(* CoDeSys 2.3.9.31 project: convertedProject.pr6 *)
(* Libraries: Standard.lib 5.6.98 11:03:02 *)

(* Task configuration *)
TASK MainTask (PRIORITY := 1, INTERVAL := T#200ms);
	MAIN();
END_TASK

(* Global variable list: Global_Variables *)
VAR_GLOBAL
	(* Контроль 0 *)
	G_IN_CTL_BTN_1: BOOL; (* Кнопка ALL *)
	G_IN_CTL_BTN_2: BOOL; (* Кнопка RESET *)
	G_OUT_CTL_ALARM_LAMP: BOOL; (* Лампа-сигнализатор *)
	G_OUT_CTL_ALARM_SOUND: BOOL; (* Динамик в ПЛК *)
	G_OUT_CTL_SOCKET_1: BOOL; (* Питание для МВВ *)

	(* Дверь *)
	G_IN_DOOR_DTR_1: BOOL; (* Сенсор открытия двери *)
	G_IN_DOOR_BTN_BELL: BOOL; (* Кнопка звонка *)
	G_OUT_DOOR_BELL: BOOL; (* Звонок *)

	(* Кухня 1 *)
	G_IN_KTN_BTN_1: BOOL; (* Выключатель основной *)
	G_IN_KTN_BTN_2: BOOL; (* Выключатель для вытяжки *)
	G_IN_KTN_DTR_1: BOOL; (* Датчик протечек *)
	G_OUT_KTN_LIGHT_1: BOOL; (* Свет основной *)
	G_OUT_KTN_LIGHT_2: BOOL; (* Свет второстепенный (подсветка) *)
	G_OUT_KTN_FAN_1: BOOL; (* Вытяжка *)

	(* Балкон *)
	G_IN_BLKN_BTN_1: BOOL; (* Выключатель *)
	G_OUT_BLKN_LIGHT_1: BOOL; (* Свет *)

	(* Гостиная *)
	G_IN_LVG_BTN_1: BOOL; (* Выключатель *)
	G_IN_LVG_BTN_2: BOOL; (* Выключатель на рабочем месте *)
	G_OUT_LVG_LIGHT_1: BOOL; (* Свет основной *)
	G_OUT_LVG_LIGHT_2: BOOL; (* Свет второстепенный *)

	(* Спальная *)
	G_IN_BDR_BTN_1: BOOL; (* Выключатель *)
	G_IN_BDR_BTN_2: BOOL; (* Выключатель над кроватью *)
	G_IN_BDR_BTN_3: BOOL; (* Выключатель над кроватью *)
	G_OUT_BDR_LIGHT_1: BOOL; (* Свет *)
	G_OUT_BDR_LIGHT_2: BOOL; (* Свет второстепенный *)
	G_OUT_BDR_LIGHT_3: BOOL; (* Свет над кроватью (торшер) *)
	G_OUT_BDR_LIGHT_4: BOOL; (* Свет над кроватью (торшер) *)

	(* Ванная большая *)
	G_IN_BMB_BTN_1: BOOL; (* Выключатель основной *)
	G_IN_BMB_BTN_2: BOOL; (* Выключатель около зеркала *)
	G_IN_BMB_DTR_1: BOOL; (* Датчик протечек *)
	G_OUT_BMB_LIGHT_1: BOOL; (* Свет основной *)
	G_OUT_BMB_LIGHT_2: BOOL; (* Свет около зеркала *)
	G_OUT_BMB_FAN_1: BOOL; (* Вытяжка *)
	G_OUT_BMB_VLV_1: BOOL; (* Вентиль *)
	G_OUT_BMB_VLV_2: BOOL; (* Вентиль *)

	(* Детская *)
	G_IN_CHLD_BTN_1: BOOL; (* Выключатель *)
	G_OUT_CHLD_LIGHT_1: BOOL; (* Свет основной *)
	G_OUT_CHLD_LIGHT_2: BOOL; (* Свет второстепенный *)

	(* Коридор *)
	G_IN_HLL_BTN_1: BOOL; (* Проходной выключатель *)
	G_IN_HLL_BTN_2: BOOL; (* Проходной выключатель *)
	G_IN_HLL_BTN_3: BOOL; (* Выключатель на зеркало *)
	G_IN_HLL_BTN_4: BOOL; (* Выключатель в шкафу *)
	G_IN_HLL_BTN_5: BOOL; (* Выключатель в шкафу *)

	G_OUT_HLL_LIGHT_1: BOOL; (* Свет основной *)
	G_OUT_HLL_LIGHT_2: BOOL; (* Свет второстепенный *)
	G_OUT_HLL_LIGHT_3: BOOL; (* Свет зеркало *)
	G_OUT_HLL_LIGHT_4: BOOL; (* Свет в шкафу *)
	G_OUT_HLL_LIGHT_5: BOOL; (* Свет в шкафу *)

	(* Ванная малая *)
	G_IN_BMS_BTN_1: BOOL; (* Выключатель *)
	G_IN_BMS_DTR_1: BOOL; (* Датчик протечек *)
	G_OUT_BMS_LIGHT_1: BOOL; (* Вытяжка *)
	G_OUT_BMS_FAN_1: BOOL; (* Вытяжка *)
	G_OUT_BMS_VLV_1: BOOL; (* Вентиль *)
	G_OUT_BMS_VLV_2: BOOL; (* Вентиль *)

	(* Розетки *)
	(* Кухня и балкон *)
	G_OUT_1_2_SOCKET_G1: BOOL; (* Общие *)
	G_OUT_1_2_SOCKET_G2: BOOL; (* Неотключаемые (холодильник)*)
	G_OUT_1_2_SOCKET_G3: BOOL; (* Посудомойка *)
	G_OUT_1_2_SOCKET_G4: BOOL; (* Плита, 380В *)
	(* Гостиная и спальня *)
	G_OUT_3_4_SOCKET_G1: BOOL; (* Общие *)
	G_OUT_3_4_SOCKET_G2: BOOL; (* Неотключаемые (компьютер) *)
	(* Ванная большая *)
	G_OUT_5_SOCKET_G1: BOOL; (* Общие *)
	G_OUT_5_SOCKET_G2: BOOL; (* Стиральная машина *)
	G_OUT_5_SOCKET_G3: BOOL; (* Резерв на бойлер и (или) баню *)
	(* Коридор и детская *)
	G_OUT_6_7_SOCKET_G1: BOOL; (* Общие *)
	G_OUT_6_7_SOCKET_G2: BOOL; (* Неотключаемые (рядом со щитком, роутер, сервер и т.п.) *)

END_VAR

(* Global variable list: TwinCAT_Import *)
VAR_GLOBAL (* DO NOT CHANGE THIS SHEET MANUALLY! *)
	PlcInVar_0	AT %QB128:	USINT;
	PlcInVar_1	AT %QB129:	USINT;
	PlcInVar_2	AT %QB130:	USINT;
	PlcInVar_3	AT %QB131:	USINT;
	PlcInVar_4	AT %QB132:	USINT;
	PlcInVar_5	AT %QB133:	USINT;
	PlcInVar_6	AT %QB134:	USINT;
	PlcInVar_7	AT %QB135:	USINT;
	PlcInVar_8	AT %QB136:	USINT;
	PlcInVar_9	AT %QB137:	USINT;
	PlcInVar_10	AT %QB138:	USINT;
	PlcInVar_11	AT %QB139:	USINT;
	PlcInVar_12	AT %QB140:	USINT;
	PlcInVar_13	AT %QB141:	USINT;
	PlcInVar_14	AT %QB142:	USINT;
	PlcInVar_15	AT %QB143:	USINT;
	PlcOutVar_0	AT %IB128:	USINT;
	PlcOutVar_1	AT %IB129:	USINT;
	PlcOutVar_2	AT %IB130:	USINT;
	PlcOutVar_3	AT %IB131:	USINT;
	PlcOutVar_4	AT %IB132:	USINT;
	PlcOutVar_5	AT %IB133:	USINT;
	PlcOutVar_6	AT %IB134:	USINT;
	PlcOutVar_7	AT %IB135:	USINT;
	PlcOutVar_8	AT %IB136:	USINT;
	PlcOutVar_9	AT %IB137:	USINT;
	PlcOutVar_10	AT %IB138:	USINT;
	PlcOutVar_11	AT %IB139:	USINT;
	PlcOutVar_12	AT %IB140:	USINT;
	PlcOutVar_13	AT %IB141:	USINT;
	PlcOutVar_14	AT %IB142:	USINT;
	PlcOutVar_15	AT %IB143:	USINT;
	Term_2_KL2408_1_Output	AT %QX0.0:	BOOL;
	Term_2_KL2408_2_Output	AT %QX0.1:	BOOL;
	Term_2_KL2408_3_Output	AT %QX0.2:	BOOL;
	Term_2_KL2408_4_Output	AT %QX0.3:	BOOL;
	Term_2_KL2408_5_Output	AT %QX0.4:	BOOL;
	Term_2_KL2408_6_Output	AT %QX0.5:	BOOL;
	Term_2_KL2408_7_Output	AT %QX0.6:	BOOL;
	Term_2_KL2408_8_Output	AT %QX0.7:	BOOL;
	Term_3_KL2408_1_Output	AT %QX1.0:	BOOL;
	Term_3_KL2408_2_Output	AT %QX1.1:	BOOL;
	Term_3_KL2408_3_Output	AT %QX1.2:	BOOL;
	Term_3_KL2408_4_Output	AT %QX1.3:	BOOL;
	Term_3_KL2408_5_Output	AT %QX1.4:	BOOL;
	Term_3_KL2408_6_Output	AT %QX1.5:	BOOL;
	Term_3_KL2408_7_Output	AT %QX1.6:	BOOL;
	Term_3_KL2408_8_Output	AT %QX1.7:	BOOL;
	Term_4_KL2408_1_Output	AT %QX2.0:	BOOL;
	Term_4_KL2408_2_Output	AT %QX2.1:	BOOL;
	Term_4_KL2408_3_Output	AT %QX2.2:	BOOL;
	Term_4_KL2408_4_Output	AT %QX2.3:	BOOL;
	Term_4_KL2408_5_Output	AT %QX2.4:	BOOL;
	Term_4_KL2408_6_Output	AT %QX2.5:	BOOL;
	Term_4_KL2408_7_Output	AT %QX2.6:	BOOL;
	Term_4_KL2408_8_Output	AT %QX2.7:	BOOL;
	Term_5_KL2408_1_Output	AT %QX3.0:	BOOL;
	Term_5_KL2408_2_Output	AT %QX3.1:	BOOL;
	Term_5_KL2408_3_Output	AT %QX3.2:	BOOL;
	Term_5_KL2408_4_Output	AT %QX3.3:	BOOL;
	Term_5_KL2408_5_Output	AT %QX3.4:	BOOL;
	Term_5_KL2408_6_Output	AT %QX3.5:	BOOL;
	Term_5_KL2408_7_Output	AT %QX3.6:	BOOL;
	Term_5_KL2408_8_Output	AT %QX3.7:	BOOL;
	Term_6_KL2408_1_Output	AT %QX4.0:	BOOL;
	Term_6_KL2408_2_Output	AT %QX4.1:	BOOL;
	Term_6_KL2408_3_Output	AT %QX4.2:	BOOL;
	Term_6_KL2408_4_Output	AT %QX4.3:	BOOL;
	Term_6_KL2408_5_Output	AT %QX4.4:	BOOL;
	Term_6_KL2408_6_Output	AT %QX4.5:	BOOL;
	Term_6_KL2408_7_Output	AT %QX4.6:	BOOL;
	Term_6_KL2408_8_Output	AT %QX4.7:	BOOL;
	Term_7_KL1408_1_Input	AT %IX0.0:	BOOL;
	Term_7_KL1408_2_Input	AT %IX0.1:	BOOL;
	Term_7_KL1408_3_Input	AT %IX0.2:	BOOL;
	Term_7_KL1408_4_Input	AT %IX0.3:	BOOL;
	Term_7_KL1408_5_Input	AT %IX0.4:	BOOL;
	Term_7_KL1408_6_Input	AT %IX0.5:	BOOL;
	Term_7_KL1408_7_Input	AT %IX0.6:	BOOL;
	Term_7_KL1408_8_Input	AT %IX0.7:	BOOL;
	Term_8_KL1408_1_Input	AT %IX1.0:	BOOL;
	Term_8_KL1408_2_Input	AT %IX1.1:	BOOL;
	Term_8_KL1408_3_Input	AT %IX1.2:	BOOL;
	Term_8_KL1408_4_Input	AT %IX1.3:	BOOL;
	Term_8_KL1408_5_Input	AT %IX1.4:	BOOL;
	Term_8_KL1408_6_Input	AT %IX1.5:	BOOL;
	Term_8_KL1408_7_Input	AT %IX1.6:	BOOL;
	Term_8_KL1408_8_Input	AT %IX1.7:	BOOL;
	Term_9_KL1408_1_Input	AT %IX2.0:	BOOL;
	Term_9_KL1408_2_Input	AT %IX2.1:	BOOL;
	Term_9_KL1408_3_Input	AT %IX2.2:	BOOL;
	Term_9_KL1408_4_Input	AT %IX2.3:	BOOL;
	Term_9_KL1408_5_Input	AT %IX2.4:	BOOL;
	Term_9_KL1408_6_Input	AT %IX2.5:	BOOL;
	Term_9_KL1408_7_Input	AT %IX2.6:	BOOL;
	Term_9_KL1408_8_Input	AT %IX2.7:	BOOL;
	Term_10_KL1408_1_Input	AT %IX3.0:	BOOL;
	Term_10_KL1408_2_Input	AT %IX3.1:	BOOL;
	Term_10_KL1408_3_Input	AT %IX3.2:	BOOL;
	Term_10_KL1408_4_Input	AT %IX3.3:	BOOL;
	Term_10_KL1408_5_Input	AT %IX3.4:	BOOL;
	Term_10_KL1408_6_Input	AT %IX3.5:	BOOL;
	Term_10_KL1408_7_Input	AT %IX3.6:	BOOL;
	Term_10_KL1408_8_Input	AT %IX3.7:	BOOL;
END_VAR

(* POU MAIN, ST *)
PROGRAM MAIN
VAR
	KTN_BTN_1 : Z_FB_DIFF_OUT_ON_LONG_AND_SHORT;
	KTN_BTN_2 : Z_FB_SINGLE_SW;

	BLKN_BTN : Z_FB_SINGLE_SW;

	LVG_BTN : Z_FB_SHORT_P_OUT1_LONG_P_OUT1_AND_OUT2;

	BDR_BTN_1 : Z_FB_SHORT_P_OUT1_LONG_P_OUT1_AND_OUT2;
	BDR_BTN_2 : Z_FB_SINGLE_SW;
	BDR_BTN_3 : Z_FB_SINGLE_SW;

	BMB_BTN_1 : Z_FB_SHRT_P_OUT1_LNG_P_OUT1_OUT2_TIMER;
	BMB_BTN_2 : Z_FB_SINGLE_SW;

	CHLD_BTN : Z_FB_SHORT_P_OUT1_LONG_P_OUT1_AND_OUT2;

	HLL_BTN_1_2 : FB_HLL;
	HLL_BTN_3 : Z_FB_SINGLE_SW_WITH_TIMER;
	HLL_BTN_4 : Z_FB_SINGLE_SW_WITH_TIMER;
	HLL_BTN_5 : Z_FB_SINGLE_SW_WITH_TIMER;

	BMS_BTN : Z_FB_SHRT_P_OUT1_LNG_P_OUT1_OUT2_TIMER;

	CTL_BTN_ALL : FB_ALL;

	IN_WS_LEFT : Z_FB_WS;
	IN_WS_RIGHT : Z_FB_WS;

	T_LONG_PRESS : TIME := t#1000ms;
	T_LIGHT_OFF : TIME := t#5000ms;
	T_FAN_OFF : TIME := t#5000ms;

	ALARM : FB_ALARM;

	ERROR : BOOL;

END_VAR
(* Основной выключатель на кухне *)
KTN_BTN_1 (IN := G_IN_KTN_BTN_1, Q1 := G_OUT_KTN_LIGHT_1, Q2 := G_OUT_KTN_LIGHT_2, TC := T_LONG_PRESS);

(* Второстепенный выключатель на кухне *)
KTN_BTN_2 (IN := G_IN_KTN_BTN_2, Q :=  G_OUT_KTN_FAN_1);

(* Выключатель на балконе *)
BLKN_BTN (IN := G_IN_BLKN_BTN_1, Q := G_OUT_BLKN_LIGHT_1);

(* Выключатели в гостиной *)
LVG_BTN (IN := G_IN_LVG_BTN_1 OR G_IN_LVG_BTN_2, Q1 := G_OUT_LVG_LIGHT_1, Q2 := G_OUT_LVG_LIGHT_2, TC := T_LONG_PRESS);

(* Выключатели в спальне *)
BDR_BTN_1 (IN := G_IN_BDR_BTN_1, Q1 := G_OUT_BDR_LIGHT_1, Q2 := G_OUT_BDR_LIGHT_2, TC := T_LONG_PRESS);
BDR_BTN_2 (IN := G_IN_BDR_BTN_2, Q := G_OUT_BDR_LIGHT_3);
BDR_BTN_3 (IN := G_IN_BDR_BTN_3, Q := G_OUT_BDR_LIGHT_4);

(* Выключатель в санузле *)
BMB_BTN_1 (IN := G_IN_BMB_BTN_1, Q1 := G_OUT_BMB_LIGHT_1, Q2 := G_OUT_BMB_FAN_1, TC := T_LONG_PRESS, TLight := T_LIGHT_OFF, TFan := T_FAN_OFF);
BMB_BTN_2 (IN := G_IN_BMB_BTN_2, Q := G_OUT_BMB_LIGHT_2);

(* Выключатели в детской *)
CHLD_BTN (IN := G_IN_CHLD_BTN_1, Q1 := G_OUT_CHLD_LIGHT_1, Q2 := G_OUT_CHLD_LIGHT_2, TC := T_LONG_PRESS);

(* Выключатель в коридоре *)
HLL_BTN_1_2 (IN := G_IN_HLL_BTN_1 OR G_IN_HLL_BTN_2, Q1 := G_OUT_HLL_LIGHT_1, Q2 := G_OUT_HLL_LIGHT_2, TC := T_LONG_PRESS);
HLL_BTN_3 (IN := G_IN_HLL_BTN_3, Q :=G_OUT_HLL_LIGHT_3, TC := T_LIGHT_OFF);
HLL_BTN_4 (IN := G_IN_HLL_BTN_4, Q :=G_OUT_HLL_LIGHT_4, TC := T_LIGHT_OFF);
HLL_BTN_5 (IN := G_IN_HLL_BTN_5, Q :=G_OUT_HLL_LIGHT_5, TC := T_LIGHT_OFF);

(* Выключатель в санузле *)
BMS_BTN (IN := G_IN_BMS_BTN_1, Q1 := G_OUT_BMS_LIGHT_1, Q2 := G_OUT_BMS_FAN_1, TC := T_LONG_PRESS, TLight := T_LIGHT_OFF, TFan := T_FAN_OFF);

(* Дверной звонок *)
(* TODO *)

(* Датчики протечек слева *)
IN_WS_LEFT(IN := G_IN_KTN_DTR_1 OR G_IN_BMS_DTR_1, RESET := G_IN_CTL_BTN_2, Q1 := G_OUT_BMS_VLV_1, Q2 := G_OUT_BMS_VLV_2, ALARM => ERROR);

(* Датчики протечек справа *)
IN_WS_RIGHT(IN := G_IN_BMB_DTR_1, RESET := G_IN_CTL_BTN_2, Q1 := G_OUT_BMB_VLV_1, Q2 := G_OUT_BMB_VLV_2, ALARM => ERROR);

(* Обработка тревоги *)
ALARM(ERROR := ERROR, Q1 := G_OUT_CTL_ALARM_LAMP, Q2 := G_OUT_CTL_ALARM_SOUND);

(* Общий выключатель *)
(* CTL_BTN_ALL(IN := G_IN_CTL_BTN_1, TC := T_LONG_PRESS); *)

(* Обработка общего выключателя *)
IF CTL_BTN_ALL.Q1 THEN

	G_OUT_KTN_LIGHT_1 := FALSE;
	G_OUT_KTN_LIGHT_2 := FALSE;
	G_OUT_KTN_FAN_1 := FALSE;

	G_OUT_BLKN_LIGHT_1 := FALSE;

	G_OUT_BMS_LIGHT_1 := FALSE;
	G_OUT_BMS_FAN_1 := FALSE;

ELSIF CTL_BTN_ALL.Q2 THEN

	G_OUT_1_2_SOCKET_G1 := FALSE;
	G_OUT_1_2_SOCKET_G3 := FALSE;
	G_OUT_1_2_SOCKET_G4 := FALSE;

	G_OUT_3_4_SOCKET_G1 := FALSE;
	G_OUT_3_4_SOCKET_G2 := FALSE;

	G_OUT_5_SOCKET_G1 := FALSE;
	G_OUT_5_SOCKET_G3 := FALSE;

	G_OUT_6_7_SOCKET_G1 := FALSE;

ELSE

	G_OUT_1_2_SOCKET_G1 := CTL_BTN_ALL.G1_STATE;
	G_OUT_1_2_SOCKET_G3 := CTL_BTN_ALL.G1_STATE;
	G_OUT_1_2_SOCKET_G4 := CTL_BTN_ALL.G1_STATE;

	G_OUT_3_4_SOCKET_G1 := CTL_BTN_ALL.G1_STATE;
	G_OUT_3_4_SOCKET_G2 := CTL_BTN_ALL.G1_STATE;

	G_OUT_5_SOCKET_G1 := CTL_BTN_ALL.G1_STATE;
	G_OUT_5_SOCKET_G3 := CTL_BTN_ALL.G1_STATE;

	G_OUT_6_7_SOCKET_G1 := CTL_BTN_ALL.G1_STATE;

END_IF;
END_PROGRAM

(* POU Z_FB_DIFF_OUT_ON_LONG_AND_SHORT, ST *)
(* Обработка длинного и короткого нажатия на два независимых выхода *)
FUNCTION_BLOCK Z_FB_DIFF_OUT_ON_LONG_AND_SHORT
VAR_INPUT
	IN : BOOL;
   	TC : TIME;
END_VAR
VAR_IN_OUT
	Q1 : BOOL;
	Q2 : BOOL;
END_VAR
VAR
	TX : TON;
	MEM1 : BOOL;
	MEM2 : BOOL;
END_VAR
TX(IN := IN, PT := TC);

IF TX.Q AND NOT MEM2 AND IN THEN
	Q2 := NOT Q2;
ELSIF NOT IN AND MEM1 AND NOT MEM2 THEN
	Q1 := NOT Q1;
END_IF;

MEM1 :=  IN;
MEM2 := TX.Q;
END_FUNCTION_BLOCK

(* POU Z_FB_SINGLE_SW, ST *)
(* Кнопка как выключатель *)
FUNCTION_BLOCK Z_FB_SINGLE_SW
VAR_INPUT
	IN: BOOL;
END_VAR
VAR_IN_OUT
	Q: BOOL;
END_VAR
VAR
	MEM : BOOL := FALSE;
END_VAR
IF IN AND NOT MEM THEN
	Q := NOT Q;
END_IF

MEM := IN;
END_FUNCTION_BLOCK

(* POU Z_FB_SHORT_P_OUT1_LONG_P_OUT1_AND_OUT2, ST *)
(* Два выхода
первый - короткое нажатие
первый и второй - длинное нажатие*)
FUNCTION_BLOCK Z_FB_SHORT_P_OUT1_LONG_P_OUT1_AND_OUT2
VAR_INPUT
	IN : BOOL;
   	TC : TIME;
END_VAR
VAR_IN_OUT
	Q1 : BOOL;
	Q2 : BOOL;
END_VAR
VAR
	TX : TON;
	MEM1, MEM2 : BOOL;
END_VAR
TX(IN := IN, PT := TC);

IF IN AND NOT MEM1 THEN
      Q1 := NOT Q1;
      IF NOT Q1 THEN
         Q2 := FALSE;
      END_IF
END_IF

IF TX.Q AND NOT MEM2 AND Q1 THEN
      Q2 := TRUE;
END_IF;

MEM1 := IN;
MEM2 := TX.Q;
END_FUNCTION_BLOCK

(* POU Z_FB_SHRT_P_OUT1_LNG_P_OUT1_OUT2_TIMER, ST *)
(* Два выхода
первый - короткое нажатие
первый и второй - длинное нажатие
при OUT2 = TRUE и длинном нажатии отключается OUT1 и OUT2, 
при OUT1 = TRUE и коротком нажатии отключается OUT1, а OUT2 отключается по таймеру
при OUT1 = TRUE OUT1 отключается по таймеру
*)
FUNCTION_BLOCK Z_FB_SHRT_P_OUT1_LNG_P_OUT1_OUT2_TIMER
VAR_INPUT
	IN : BOOL;
   	TC : TIME;
	TFan : TIME;
	TLight : TIME;
END_VAR
VAR_IN_OUT
	Q1 : BOOL;
	Q2 : BOOL;
END_VAR
VAR
	TX : TON;
	TPFanInst : TOF;
	TPLightInst : TP;
	MEM1, MEM2 : BOOL;
END_VAR
TX(IN := IN, PT := TC);

IF TX.Q AND NOT MEM2 AND IN THEN
	Q1 := NOT Q1;
	Q2 := NOT Q2;
ELSIF NOT IN AND MEM1 AND NOT MEM2 THEN
	Q1 := NOT Q1;
END_IF

TPFanInst(PT := TFan, IN := Q1);
IF Q2 AND NOT TPFanInst.Q THEN
	Q2 := TPFanInst.Q;
END_IF

TPLightInst(PT := TLight, IN := Q1);
IF Q1 AND NOT TPLightInst.Q THEN
	Q1 := TPLightInst.Q;
	Q2 := TPLightInst.Q;
END_IF

(*AND NOT MEM2 AND IN THEN
	Q2 := NOT Q2;
	Q1 := NOT Q1;
ELSIF NOT IN AND MEM1 THEN
	(*IF NOT MEM2 AND NOT Q2 THEN*)
		Q1 := NOT Q1;
	ELSIF NOT MEM2 AND MEM1 THEN
		Q2 := NOT Q2;
	END_IF;
END_IF;*)

MEM1 :=  IN;
MEM2 := TX.Q;
END_FUNCTION_BLOCK

(* POU FB_HLL, ST *)
FUNCTION_BLOCK FB_HLL
VAR_INPUT
	IN : BOOL;
   	TC : TIME;
END_VAR
VAR_IN_OUT
	Q1 : BOOL;
	Q2 : BOOL;
END_VAR
VAR
	TX : TON;
	MEM1, MEM2 : BOOL;
END_VAR
TX(IN := IN, PT := TC);

IF TX.Q AND NOT MEM2 AND IN THEN
	Q2 := NOT Q2;
ELSIF NOT IN AND MEM1 THEN
	IF NOT MEM2 AND NOT Q2 THEN
		Q1 := NOT Q1;
	ELSIF NOT MEM2 AND MEM1 THEN
		Q2 := NOT Q2;
	END_IF;
END_IF;

MEM1 :=  IN;
MEM2 := TX.Q;
END_FUNCTION_BLOCK

(* POU Z_FB_SINGLE_SW_WITH_TIMER, ST *)
(* Кнопка как выключатель c таймером на отключение *)
FUNCTION_BLOCK Z_FB_SINGLE_SW_WITH_TIMER
VAR_INPUT
	IN: BOOL;
	TC : TIME;
END_VAR
VAR_IN_OUT
	Q: BOOL;
END_VAR
VAR
	MEM : BOOL := FALSE;
	TPInst : TP;
END_VAR
IF IN AND NOT MEM THEN
	Q := NOT Q;
END_IF

TPInst(PT := TC, IN := Q);
IF Q AND NOT TPInst.Q THEN
	Q := TPInst.Q;
END_IF

MEM := IN;
END_FUNCTION_BLOCK

(* POU FB_ALL, ST *)
FUNCTION_BLOCK FB_ALL
VAR_INPUT
	IN: BOOL;
	TC : TIME;
END_VAR
VAR_OUTPUT
	Q1: BOOL := FALSE;
	Q2: BOOL := FALSE;
	G1_STATE: BOOL := TRUE;
END_VAR
VAR
	TX: TON;
	MEM: BOOL;
END_VAR
TX(IN := IN, PT := TC);

IF IN THEN
	IF TX.Q AND NOT MEM THEN
		Q2 := TRUE;
	ELSIF TX.Q AND MEM THEN
		G1_STATE := FALSE;
	ELSIF NOT MEM THEN
		Q1 := TRUE;
		G1_STATE := TRUE;
	END_IF;
ELSE
	Q1 := FALSE;
	Q2 := FALSE;
END_IF;

MEM := TX.Q;
END_FUNCTION_BLOCK

(* POU Z_FB_WS, ST *)
(* Слушаем сенсоры *)
FUNCTION_BLOCK Z_FB_WS
VAR_INPUT
	IN : BOOL;
	RESET : BOOL;
END_VAR
VAR_IN_OUT
	Q1 : BOOL;
	Q2 : BOOL;
END_VAR
VAR_OUTPUT
	ALARM : BOOL := FALSE;
END_VAR
VAR
	MEM : BOOL := FALSE;
END_VAR
IF IN THEN
	Q1 := TRUE;
	Q2 := TRUE;
	ALARM := TRUE;
ELSIF RESET THEN
	Q1 := FALSE;
	Q2 := FALSE;
	ALARM := FALSE;
END_IF

MEM := IN;
END_FUNCTION_BLOCK

(* POU FB_ALARM, ST *)
FUNCTION_BLOCK FB_ALARM
VAR_INPUT
	ERROR : BOOL;
END_VAR
VAR_IN_OUT
	Q1 : BOOL;
	Q2 : BOOL;
END_VAR
VAR
	tProcessTime : TIME;
	tmTimer : TON := (PT:= T#2s);
	Q: BOOL;
END_VAR
IF ERROR THEN
	tmTimer(IN := tProcessTime < T#2S, ET => tProcessTime);
	Q := tProcessTime < T#1S;
ELSE
	Q := FALSE;
END_IF;
Q1 := Q;
Q2 := Q;
END_FUNCTION_BLOCK

(* Visualisation TC_VISU
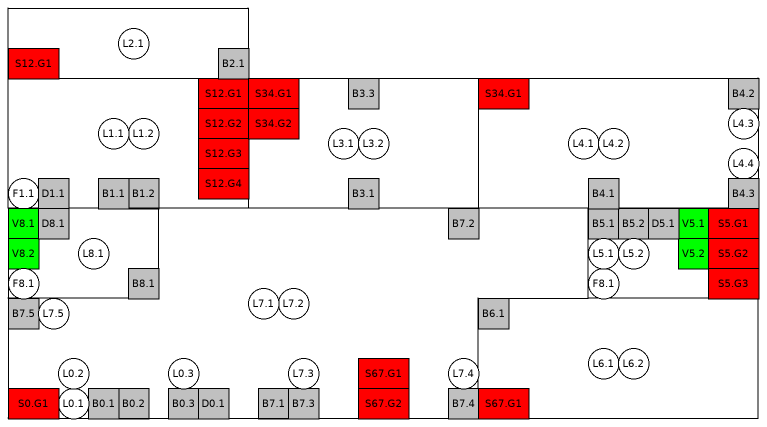
rectangle at (130,180)-(161,211): text "B1.2"; alarm colour if .G_IN_KTN_BTN_2; taps .G_IN_KTN_BTN_2
ellipse at (130,120)-(161,151): text "L1.2"; alarm colour if .G_OUT_KTN_LIGHT_2
ellipse at (100,120)-(131,151): text "L1.1"; alarm colour if .G_OUT_KTN_LIGHT_1
rectangle at (260,390)-(291,421): text "B7.1"; alarm colour if .G_IN_HLL_BTN_1; taps .G_IN_HLL_BTN_1
rectangle at (450,210)-(481,241): text "B7.2"; alarm colour if .G_IN_HLL_BTN_2; taps .G_IN_HLL_BTN_2
rectangle at (120,390)-(151,421): text "B0.2"; alarm colour if .G_IN_CTL_BTN_2; taps .G_IN_CTL_BTN_2
ellipse at (10,180)-(41,211): text "F1.1"; alarm colour if .G_OUT_KTN_FAN_1
rectangle at (200,80)-(251,111): text "S12.G1"; alarm colour if .G_OUT_1_2_SOCKET_G1
rectangle at (200,110)-(251,141): text "S12.G2"; alarm colour if .G_OUT_1_2_SOCKET_G2
rounded rectangle at (40,180)-(71,211): text "D1.1"; alarm colour if .G_IN_KTN_DTR_1; taps .G_IN_KTN_DTR_1
rectangle at (90,390)-(121,421): text "B0.1"; alarm colour if .G_IN_CTL_BTN_1; taps .G_IN_CTL_BTN_1
rectangle at (10,210)-(41,241): text "V8.1"; alarm colour if .G_OUT_BMS_VLV_1
rectangle at (10,240)-(41,271): text "V8.2"; alarm colour if .G_OUT_BMS_VLV_2
rectangle at (350,180)-(381,211): text "B3.1"; alarm colour if .G_IN_LVG_BTN_1; taps .G_IN_LVG_BTN_1
rectangle at (130,270)-(161,301): text "B8.1"; alarm colour if .G_IN_BMS_BTN_1; taps .G_IN_BMS_BTN_1
rectangle at (590,210)-(621,241): text "B5.1"; alarm colour if .G_IN_BMB_BTN_1; taps .G_IN_BMB_BTN_1
rectangle at (680,210)-(711,241): text "V5.1"; alarm colour if .G_OUT_BMB_VLV_1
rectangle at (680,240)-(711,271): text "V5.2"; alarm colour if .G_OUT_BMB_VLV_2
rectangle at (620,210)-(651,241): text "B5.2"; alarm colour if .G_IN_BMB_BTN_2; taps .G_IN_BMB_BTN_2
rounded rectangle at (40,210)-(71,241): text "D8.1"; alarm colour if .G_IN_BMS_DTR_1; taps .G_IN_BMS_DTR_1
rectangle at (100,180)-(131,211): text "B1.1"; alarm colour if .G_IN_KTN_BTN_1; taps .G_IN_KTN_BTN_1
rectangle at (450,390)-(481,421): text "B7.4"; alarm colour if .G_IN_HLL_BTN_4; taps .G_IN_HLL_BTN_4
rectangle at (10,300)-(41,331): text "B7.5"; alarm colour if .G_IN_HLL_BTN_5; taps .G_IN_HLL_BTN_5
rectangle at (350,80)-(381,111): text "B3.3"; alarm colour if .G_IN_LVG_BTN_2; taps .G_IN_LVG_BTN_2
ellipse at (120,30)-(151,61): text "L2.1"; alarm colour if .G_OUT_BLKN_LIGHT_1
rectangle at (220,50)-(251,81): text "B2.1"; alarm colour if .G_IN_BLKN_BTN_1; taps .G_IN_BLKN_BTN_1
rectangle at (290,390)-(321,421): text "B7.3"; alarm colour if .G_IN_HLL_BTN_3; taps .G_IN_HLL_BTN_3
rectangle at (170,390)-(201,421): text "B0.3"; alarm colour if .G_IN_DOOR_BTN_BELL; taps .G_IN_DOOR_BTN_BELL
ellipse at (330,130)-(361,161): text "L3.1"; alarm colour if .G_OUT_LVG_LIGHT_1
ellipse at (360,130)-(391,161): text "L3.2"; alarm colour if .G_OUT_LVG_LIGHT_2
rectangle at (590,180)-(621,211): text "B4.1"; alarm colour if .G_IN_BDR_BTN_1; taps .G_IN_BDR_BTN_1
rectangle at (730,80)-(761,111): text "B4.2"; alarm colour if .G_IN_BDR_BTN_2; taps .G_IN_BDR_BTN_2
ellipse at (730,110)-(761,141): text "L4.3"; alarm colour if .G_OUT_BDR_LIGHT_3
ellipse at (730,150)-(761,181): text "L4.4"; alarm colour if .G_OUT_BDR_LIGHT_4
rectangle at (730,180)-(761,211): text "B4.3"; alarm colour if .G_IN_BDR_BTN_3; taps .G_IN_BDR_BTN_3
ellipse at (570,130)-(601,161): text "L4.1"; alarm colour if .G_OUT_BDR_LIGHT_1
ellipse at (600,130)-(631,161): text "L4.2"; alarm colour if .G_OUT_BDR_LIGHT_2
rounded rectangle at (650,210)-(681,241): text "D5.1"; alarm colour if .G_IN_BMB_DTR_1; taps .G_IN_BMB_DTR_1
rectangle at (480,300)-(511,331): text "B6.1"; alarm colour if .G_IN_CHLD_BTN_1; taps .G_IN_CHLD_BTN_1
ellipse at (590,350)-(621,381): text "L6.1"; alarm colour if .G_OUT_CHLD_LIGHT_1
ellipse at (620,350)-(651,381): text "L6.2"; alarm colour if .G_OUT_CHLD_LIGHT_2
ellipse at (280,290)-(311,321): text "L7.2"; alarm colour if .G_OUT_HLL_LIGHT_2
ellipse at (250,290)-(281,321): text "L7.1"; alarm colour if .G_OUT_HLL_LIGHT_1
ellipse at (40,300)-(71,331): text "L7.5"; alarm colour if .G_OUT_HLL_LIGHT_5
ellipse at (290,360)-(321,391): text "L7.3"; alarm colour if .G_OUT_HLL_LIGHT_3
ellipse at (450,360)-(481,391): text "L7.4"; alarm colour if .G_OUT_HLL_LIGHT_4
ellipse at (60,390)-(91,421): text "L0.1"; alarm colour if .G_OUT_CTL_ALARM_LAMP
rounded rectangle at (200,390)-(231,421): text "D0.1"; alarm colour if .G_IN_DOOR_DTR_1; taps .G_IN_DOOR_DTR_1
ellipse at (80,240)-(111,271): text "L8.1"; alarm colour if .G_OUT_BMS_LIGHT_1
ellipse at (10,270)-(41,301): text "F8.1"; alarm colour if .G_OUT_BMS_FAN_1
ellipse at (590,270)-(621,301): text "F8.1"; alarm colour if .G_OUT_BMB_FAN_1
ellipse at (60,360)-(91,391): text "L0.2"; alarm colour if .G_OUT_CTL_ALARM_SOUND
ellipse at (590,240)-(621,271): text "L5.1"; alarm colour if .G_OUT_BMB_LIGHT_1
ellipse at (620,240)-(651,271): text "L5.2"; alarm colour if .G_OUT_BMB_LIGHT_2
ellipse at (170,360)-(201,391): text "L0.3"; alarm colour if .G_OUT_DOOR_BELL
rectangle at (200,140)-(251,171): text "S12.G3"; alarm colour if .G_OUT_1_2_SOCKET_G3
rectangle at (10,50)-(61,81): text "S12.G1"; alarm colour if .G_OUT_1_2_SOCKET_G1
rectangle at (200,170)-(251,201): text "S12.G4"; alarm colour if .G_OUT_1_2_SOCKET_G4
rectangle at (250,80)-(301,111): text "S34.G1"; alarm colour if .G_OUT_3_4_SOCKET_G1
rectangle at (250,110)-(301,141): text "S34.G2"; alarm colour if .G_OUT_3_4_SOCKET_G2
rectangle at (710,210)-(761,241): text "S5.G1"; alarm colour if .G_OUT_5_SOCKET_G1
rectangle at (710,240)-(761,271): text "S5.G2"; alarm colour if .G_OUT_5_SOCKET_G2
rectangle at (710,270)-(761,301): text "S5.G3"; alarm colour if .G_OUT_5_SOCKET_G3
rectangle at (480,80)-(531,111): text "S34.G1"; alarm colour if .G_OUT_3_4_SOCKET_G1
rectangle at (360,360)-(411,391): text "S67.G1"; alarm colour if .G_OUT_6_7_SOCKET_G1
rectangle at (360,390)-(411,421): text "S67.G2"; alarm colour if .G_OUT_6_7_SOCKET_G2
rectangle at (10,390)-(61,421): text "S0.G1"; alarm colour if .G_OUT_CTL_SOCKET_1
rectangle at (480,390)-(531,421): text "S67.G1"; alarm colour if .G_OUT_6_7_SOCKET_G1
9 more shapes without text or variables
*)
